Fanuc KAREL source: kf00037.KL

-- PROVISIONAL review KL for V1013-1; original PC SHA256 4a3872cc0d2d79bd4c17ec4a58600c5f0adbb7bfc6477ec635b07796c9546563
-- Incomplete behavior may be omitted. Consult companion uncertainty JSON. Do not deploy.
PROGRAM KF00037
%NOLOCKGROUP
VAR
  I : INTEGER
  J : INTEGER
  X : REAL
  Y : REAL
  B : BOOLEAN
  C : BOOLEAN
  TXT : STRING[80]
  TXT2 : STRING[80]
  STATUS : INTEGER
-- UNRESOLVED_DECL AI type=002010
-- UNRESOLVED_DECL BI type=002010
-- UNRESOLVED_DECL P type=000102
-- UNRESOLVED_DECL JP type=000199
-- UNRESOLVED_DECL PF type=000101
-- UNRESOLVED_DECL V1 type=000013
-- UNRESOLVED_DECL V2 type=000013
BEGIN
  -- UNRESOLVED_PC offsets 5-23; opcodes 2E,22,2E,33,35
  -- UNRESOLVED_PC offsets 28-47; opcodes 22,2E,33,34,23
  -- UNRESOLVED_PC offsets 52-56; opcodes 7F
END KF00037
